{attribute 'GeneratedUsingTerminal: EK1122-0000-0018'}
{attribute addProperty VendorId "#x00000002"}
{attribute addProperty BoxType "EK1122-0000-0018"}
{attribute addProperty Description "EK1122 2 port EtherCAT junction"}
{attribute addProperty Physics "KYKY"}
{attribute addProperty Id "InfoDataAT %I*InfoData_6F19DB2B2"}
{attribute addProperty CRC "532711307"}
{attribute addProperty Size "2"}
TYPE EK1122_1FC0878B EXTENDS TcoIo.EtcSlaveTerminalBase_947E5A46 :
STRUCT
	{attribute addProperty Name "InfoData"}
	InfoData : TcoIo.InfoData_6F19DB2B;
END_STRUCT
END_TYPE

(* stored: Version 1.2.0.0
   DUT EK1122_1FC0878B: Id {d6d9a445-b6a8-4831-bc3f-dac949fc58b9} *)
